FUNCTION CurrentToKw : REAL
VAR_INPUT
	Current		: REAL;
	linevoltage	: REAL;
END_VAR

IF linevoltage > 100 THEN
	CurrentToKw := (Current * linevoltage * 1.73) / 1000;
ELSE
	CurrentToKw := (Current * 400 * 1.73) / 1000;
END_IF

END_FUNCTION

(* stored: Version 1.1.0.1, ProductVersion 3.1.4026.18
   POU CurrentToKw: Id {5e80c638-b1c0-44a1-8017-938fc15e25c4}, SpecialFunc None *)
